FUNCTION_BLOCK FB_AbfullModul
VAR_INPUT
    bEnable     : BOOL;
    bExecute    : BOOL; 
	bBandSens1 	: BOOL;   
    bBandSens2 	: BOOL; 
	bBandSens3 	: BOOL; 
	bBandSens4 	: BOOL; 
 	bEinzelSens1: BOOL;
	bEinzelSens2: BOOL;
	bEinzelSens3: BOOL;
	nLagerIndex : INT;
END_VAR

VAR_OUTPUT
	//Vereinzelungsoutputs
	bGate1 : BOOL;
    bGate2 : BOOL;
	//Transportoutputs
	bStopper1 : BOOL;
    bStopper2 : BOOL;
    bStopper3 : BOOL;
    eState      : eBetriebszustand;
END_VAR

VAR
    fbVereinzelung      : FB_Vereinzelung;
    fbDispenser1         : FB_Dispenser;
	fbDispenser2         : FB_Dispenser;
	fbDispenser3         : FB_Dispenser;
    fbTransport    		: FB_Transport;
	
	fTrigBandSens4 : f_TRIG; 
	bBandSens4Rise  : BOOL;
	
    nState : INT := 0;
	nStation : INT;
	
	
END_VAR

VAR_IN_OUT
    axFoerderband : Axis_Ref;
    axDispenser1    : Axis_Ref;
	axDispenser2    : Axis_Ref;
	axDispenser3    : Axis_Ref;
   // axManipulator : Axis_Ref;
END_VAR

fbVereinzelung(
	bEnable:= bEnable, 
	bExecute:=  , 
	bSensor1:= bEinzelSens1, 
	bSensor2:= bEinzelSens2 , 
	bSensor3:= bEinzelSens3 , 
	bSensor4:= bBandSens1 , 
	bGate1=> bGate1 , 
	bGate2=> bGate2, 
	eState=> );
	
fbTransport(
	bEnable:= bEnable, 
	bExecute:= , 
	nStation:= nStation, 
	bSens1:= bBandSens1, 
	bSens2:= bBandSens2, 
	bSens3:= bBandSens3 , 
	bSens4:= bBandSens4, 
	eState=> , 
	bStopper1=> bStopper1, 
	bStopper2=> bStopper2, 
	bStopper3=> bStopper3, 
	ax:= axFoerderband);
	
fbDispenser1(
	bEnable:= bEnable, 
	bExecute:=, 
	rDistance:= , 
	eState=> , 
	ax:= axDispenser1);
	
fbDispenser2(
	bEnable:= bEnable, 
	bExecute:=, 
	rDistance:= , 
	eState=> , 
	ax:= axDispenser2);
	
fbDispenser3(
	bEnable:= bEnable, 
	bExecute:= , 
	rDistance:= , 
	eState=> , 
	ax:= axDispenser3);
	
	
CASE nState OF
	0: // OFF
	eState := eBetriebszustand.Off;
	fbVereinzelung.bEnable := FALSE;
	fbVereinzelung.bExecute := FALSE;
	fbTransport.bEnable := FALSE;
	fbTransport.bExecute := FALSE;
	fbDispenser1.bEnable := FALSE;
	fbDispenser2.bEnable := FALSE;
	fbDispenser3.bEnable := FALSE;
	fbDispenser1.bExecute := FALSE;
	fbDispenser2.bExecute := FALSE;
	fbDispenser3.bExecute := FALSE;
	
	
	IF bEnable THEN
		nState := 10;
	END_IF
	
	10: // INIT
	
	eState := eBetriebszustand.Init;
	fbVereinzelung.bEnable := TRUE;
	fbVereinzelung.bExecute := FALSE;
	fbTransport.bEnable := TRUE;
	fbTransport.bExecute := FALSE;
	fbDispenser1.bEnable := TRUE;
	fbDispenser2.bEnable := TRUE;
	fbDispenser3.bEnable := TRUE;
	fbDispenser1.bExecute := FALSE;
	fbDispenser2.bExecute := FALSE;
	fbDispenser3.bExecute := FALSE;
	
	IF fbVereinzelung.eState = eBetriebszustand.Ready AND fbTransport.eState = eBetriebszustand.Ready AND fbDispenser1.eState = eBetriebszustand.Ready AND fbDispenser2.eState = eBetriebszustand.Ready AND fbDispenser3.eState = eBetriebszustand.Ready THEN
		nState := 20;
	END_IF
	
	20: // READY
	eState := eBetriebszustand.Ready;
	fbVereinzelung.bEnable := TRUE;
	fbVereinzelung.bExecute := FALSE;
	fbTransport.bEnable := TRUE;
	fbTransport.bExecute := FALSE;
	fbDispenser1.bEnable := TRUE;
	fbDispenser2.bEnable := TRUE;
	fbDispenser3.bEnable := TRUE;
	fbDispenser1.bExecute := FALSE;
	fbDispenser2.bExecute := FALSE;
	fbDispenser3.bExecute := FALSE;
	
	IF bExecute THEN
		nState := 30;
	END_IF
	
	30: //Production
	eState := eBetriebszustand.Production;
	fbVereinzelung.bExecute := TRUE;
	fbTransport.bExecute := TRUE;
	fbDispenser1.bExecute := FALSE;
	fbDispenser2.bExecute := FALSE;
	fbDispenser3.bExecute := FALSE;
	nStation := 1;
	
	IF fbVereinzelung.eState = eBetriebszustand.Done AND fbTransport.eState = eBetriebszustand.Done THEN
		nState := 31;
	END_IF
	
	31: // 1st Dispenser
	nStation := 1;
	fbDispenser1.bExecute := TRUE;
	fbVereinzelung.bExecute := FALSE;
	fbTransport.bExecute := FALSE;
	
	IF fbDispenser1.eState = eBetriebszustand.Done THEN
		nState := 32;
	END_IF
	
	32: // Bewegung zu Station 2
	nStation := 2;
	fbTransport.bExecute := TRUE;
	fbDispenser1.bExecute := FALSE;
	
	IF fbTransport.eState = eBetriebszustand.Done THEN
		nState := 33;
	END_IF
	
	33: // 2nd Dispenser
	
	fbDispenser2.bExecute := TRUE;
	fbTransport.bExecute := FALSE;
	
	IF fbDispenser2.eState = eBetriebszustand.Done THEN
		nState := 34;
	END_IF
	
	34: //Bewegung zu Station 3
	nStation := 3;
	fbTransport.bExecute := TRUE;
	fbDispenser2.bExecute := FALSE;
	
	IF fbTransport.eState = eBetriebszustand.Done THEN
		nState := 35;
	END_IF
	
	35: //3rd Dispenser
	fbTransport.bExecute := FALSE;
	fbDispenser3.bExecute := TRUE;
	
	IF fbDispenser3.eState = eBetriebszustand.Done THEN
		nState := 36;
	END_IF
	
	36: // Bewegung zu Abholstation
	nStation := 4;
	fbDispenser3.bExecute := FALSE;
	fbTransport.bExecute := TRUE;
	
	IF fbTransport.eState = eBetriebszustand.Done THEN
		nState := 40;
	END_IF
	
	40: //DONE
	eState := eBetriebszustand.Done;
	fbTransport.bExecute := FALSE;
	
	
	IF NOT bExecute THEN
		nState := 20;
	END_IF
	
	
END_CASE

END_FUNCTION_BLOCK

(* stored: Version 1.1.0.1, ProductVersion 3.1.4024.15
   POU FB_Abfullmodul: Id {2b61e3bd-8094-4055-9b51-7961cdd11497}, SpecialFunc None *)
